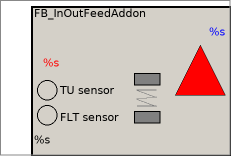
VISUALIZATION V_InOutFeedAddon  // 231x156
VAR_IN_OUT
	{attribute 'VAR_IN_OUT_AS_POINTER'}
	fbFunction		: FB_InOutFeedAddon;	
END_VAR
    Rectangle (31,6 200x150)
    Label (31,6 199x15), "FB_InOutFeedAddon"
    Rectangle (31,130 199x20), "%s", text variable: fbFunction.ConfigFunction.FunctionName
    Rectangle (40,53 160x20), "%s", text variable: fbFunction.ZoneData[1].ErrorData.Error.ErrorCode.Conv, invisible if: fbFunction.FunctionData.ErrorData.Error.ErrorCode.Conv = 0
    Polygon (175,95) (200,45) (225,95) (210,95) (190,95), invisible if: fbFunction.FunctionData.ErrorData.ErrorState = E_ErrorState.OPERATIONAL
    Rectangle (68,22 160x20), "%s", text variable: fbFunction.InOutFeedState.eState
    Ellipse (37,80 20x20), colour toggle: fbFunction.Inputs.HW.TUSensor
    Label (57,83 92x15), "TU sensor"
    Ellipse (37,105 20x20), colour toggle: fbFunction.Inputs.HW.FLTSensor
    Label (57,110 92x15), "FLT sensor"
    Polyline (156,90) (137,90) (156,97) (137,99) (156,106) (137,106), colour toggle: fbFunction.HW_Outputs.Drive_Run_UpDown, invisible if: NOT fbFunction.Settings.LiftEnabled
    Rectangle (134,111 26x12), tooltip "Lower lift sensor", colour toggle: fbFunction.HW_Inputs.Sensor_Pos_Down, invisible if: NOT fbFunction.Settings.LiftEnabled
    Rectangle (134,73 26x12), tooltip "Upper lift sensor", colour toggle: fbFunction.HW_Inputs.Sensor_Pos_Up, invisible if: NOT fbFunction.Settings.LiftEnabled
END_VISUALIZATION

(* stored: Version 1.1.0.1, ProductVersion 3.1.4024.9
   Visu V_InOutFeedAddon: Id {ecb19888-b3d6-4124-ac54-f6f53e7c0b94} *)
